{attribute 'qualified_only'}
VAR_GLOBAL
	fCyclicTime : LREAL := 0.01; 
	fPistonScale : LREAL :=100;
	fPistonPosMin : LREAL :=0;
	fPistonPosMax : LREAL :=1;
END_VAR

(* stored: Version 1.1.0.1, ProductVersion 3.1.4024.10
   GVL Parameters: Id {295e633e-08d5-4bd4-b4f1-5e6cf87cc055} *)
